SUBAPPLICATION Uebung_012c (* String Input und Speichern (WIP) *)
  (* Standard: 61499-2; Description: Copyright (c) 2023 Meisterschulen am Ostbahnhof This program and the accompanying materials are made available under the terms of the Eclipse Public License 2.0 which is available at https://www.eclipse.org/legal/epl-2.0/ SPDX-License-Identifier: EPL-2.0 *)
  (* Version 1.0, 2023-10-23, Franz Höpfinger, Meisterschulen am Ostbahnhof *)
  PACKAGE Uebungen;
  IMPORT Uebungen::const::NVS::NVS_Keys::KEY_S1_STORE;
  IMPORT Uebungen::const::NVS::NVS_Keys::SECTION_S1_STORE;
  IMPORT Uebungen::const::UT::DefaultPool::InputNumber_I1;
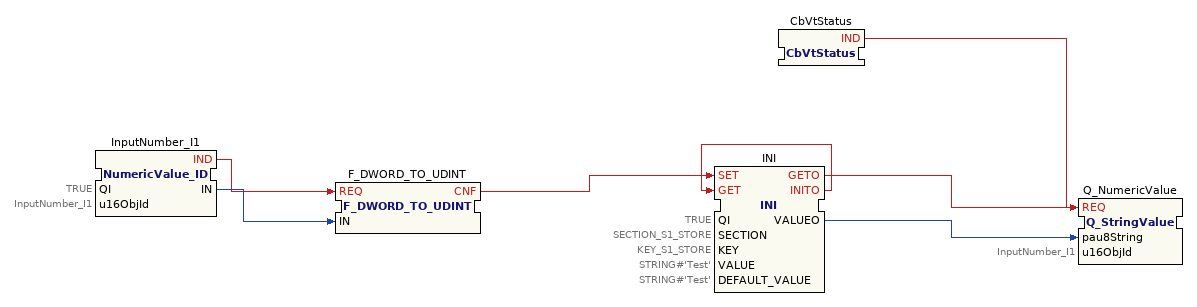
  FBS
    F_DWORD_TO_UDINT : iec61131::conversion::F_DWORD_TO_UDINT;
    InputNumber_I1 : isobus::UT::io::NumericValue::NumericValue_ID(QI := TRUE, u16ObjId := InputNumber_I1);
    INI : eclipse4diac::storage::INI(QI := TRUE, SECTION := SECTION_S1_STORE, KEY := KEY_S1_STORE, VALUE := STRING#'Test', DEFAULT_VALUE := STRING#'Test');
    Q_NumericValue : isobus::UT::Q::Q_StringValue(u16ObjId := InputNumber_I1);
    CbVtStatus : isobus::UT::status::CbVtStatus;
  END_FBS
  EVENT_CONNECTIONS
    InputNumber_I1.IND TO F_DWORD_TO_UDINT.REQ;
    F_DWORD_TO_UDINT.CNF TO INI.SET;
    INI.GETO TO Q_NumericValue.REQ;
    CbVtStatus.IND TO Q_NumericValue.REQ;
    INI.INITO TO INI.GET;
  END_CONNECTIONS
  DATA_CONNECTIONS
    InputNumber_I1.IN TO F_DWORD_TO_UDINT.IN;
    INI.VALUEO TO Q_NumericValue.pau8String;
  END_CONNECTIONS
END_SUBAPPLICATION
